PROGRAM MAIN
VAR
	var01		:	INT;
END_VAR

GVL01.var01 := 1;
GVL02.var01 := 2;
var01 := 3;

END_PROGRAM

(* stored: Version 1.1.0.1, ProductVersion 3.1.4020.6
   POU MAIN: Id {b180a901-9060-4304-b58a-988ceafe4550}, SpecialFunc None *)
